// File: DB_Plc_ManualMechAux.scl
DATA_BLOCK "DB_Plc_ManualMechAux"
{ S7_Optimized_Access := 'TRUE' }

VAR
    LastCommitSeen  : ARRAY[0..255] OF UDINT;   // PLC зберігає тут останній оброблений commit
    LastResultCode  : ARRAY[0..255] OF USINT;   // 0=OK, інше=reject (для діагностики)

    // Для розподіленої обробки (chunked processing)
    //ProcessingIndex : INT := 0;      // поточний індекс обробки
    //SlotsPerCycle   : INT := 32;     // кількість слотів за цикл (можна налаштувати)
END_VAR

BEGIN
END_DATA_BLOCK